{attribute 'GeneratedUsingTerminal: EK1122-0000-0018'}
{attribute addProperty BoxType "EK1122-0000-0018"}
{attribute addProperty Id "Beckhoff_EM7xxxsub_EK1100EK1100_AB5A94672"}
{attribute addProperty CRC "819138044"}
{attribute addProperty Size "2"}
TYPE Beckhoff_EM7xxxEK1122_30D30DFC EXTENDS EK1122_AB5A9467 :
STRUCT
	{attribute addProperty Name "Beckhoff_EM7xxxsub_EK1100"}
	Beckhoff_EM7xxxsub_EK1100 : EK1100_AB5A9467;
END_STRUCT
END_TYPE

(* stored: Version 1.2.0.0, ProductVersion 3.1.4024.9
   DUT Beckhoff_EM7xxxEK1122_30D30DFC: Id {55d62b7b-5262-4e22-9125-3643ebe86ad3} *)
